// TIA Portal V18 export
VAR_GLOBAL   // PLC tag table "Cabinet_1"
   Sz1_Button_LED_ST25_ST26 AT %Q1100.0 : Bool;
   Sz1_Button_LED_ST26_ST27 AT %Q1100.1 : Bool;
   Sz1_Button_LED_ST24_ST23 AT %Q1100.2 : Bool;
   Sz1_Button_LED_ST23_ST22 AT %Q1100.3 : Bool;
   Sz1_Button_LED_Hyd_Up AT %Q1100.4 : Bool;
   Sz1_Button_LED_Hyd_Down AT %Q1100.5 : Bool;
   Sz1_Button_LED_Air_Up AT %Q1100.6 : Bool;
   Sz1_Button_LED_Air_Down AT %Q1100.7 : Bool;
   Sz1_Button_LED_Wibration AT %Q1101.0 : Bool;
   Sz1_Button_LED_SS_Down AT %Q1101.1 : Bool;
   Sz1_Button_LED_SS_Up AT %Q1101.2 : Bool;
   Sz1_Button_LED_SS_Drive_ST25 AT %Q1101.3 : Bool;
   Sz1_Button_LED_SS_Drive_ST24 AT %Q1101.4 : Bool;
   Sz1_Button_LED_SS_Drive_ST17 AT %Q1101.5 : Bool;
   Sz1_Button_LED_SS_Drive_ST14 AT %Q1101.6 : Bool;
   Reserved AT %Q1101.7 : Bool;
   Sz1_St25_SenA AT %I1100.0 : Bool;
   Sz1_St25_SenB AT %I1100.1 : Bool;
   Sz1_St25_SenC AT %I1100.2 : Bool;
   Sz1_St25_SenD AT %I1100.3 : Bool;
   Sz1_St26_SenA AT %I1100.4 : Bool;
   Sz1_St26_SenB AT %I1100.5 : Bool;
   Sz1_St26_SenC AT %I1100.6 : Bool;
   Sz1_St26_SenD AT %I1100.7 : Bool;
   Sz1_St23_SenA AT %I1101.0 : Bool;
   Sz1_St23_SenB AT %I1101.1 : Bool;
   Sz1_St23_SenC AT %I1101.2 : Bool;
   Sz1_St23_SenD AT %I1101.3 : Bool;
   Sz1_St24_SenA AT %I1101.4 : Bool;
   Sz1_St24_SenB AT %I1101.5 : Bool;
   Sz1_St24_SenC AT %I1101.6 : Bool;
   Sz1_St24_SenD AT %I1101.7 : Bool;
   Sz1_Button_ST25_ST26 AT %I1102.0 : Bool;
   Sz1_Button_ST26_ST27 AT %I1102.1 : Bool;
   Sz1_Button_ST24_ST23 AT %I1102.2 : Bool;
   Sz1_Button_ST23_ST22 AT %I1102.3 : Bool;
   Sz1_Button_Hyd_Up AT %I1102.4 : Bool;
   Sz1_Button_Hyd_Down AT %I1102.5 : Bool;
   Sz1_Button_Air_Up AT %I1102.6 : Bool;
   Sz1_Button_Air_Down AT %I1102.7 : Bool;
   Sz1_Button_Wibration AT %I1103.0 : Bool;
   Sz1_Button_SS_Down AT %I1103.1 : Bool;
   Sz1_Button_SS_Up AT %I1103.2 : Bool;
   Sz1_Button_SS_Drive_ST25 AT %I1103.3 : Bool;
   Sz1_Button_SS_Drive_ST24 AT %I1103.4 : Bool;
   Sz1_Button_SS_Drive_ST17 AT %I1103.5 : Bool;
   Sz1_Button_SS_Drive_ST14 AT %I1103.6 : Bool;
   "Reserved(1)" AT %I1103.7 : Bool;
   Sz1_Button_Wib_ST25 AT %I1104.0 : Bool;
   Sz1_Button_Wib_ST24 AT %I1104.1 : Bool;
   Sz1_Button_Wib_ST23 AT %I1104.2 : Bool;
   Sz1_Button_Centering_ST23 AT %I1104.3 : Bool;
   Sz1_Button_Centering_ST22 AT %I1104.4 : Bool;
   "Reserved(2)" AT %I1104.5 : Bool;
   "Reserved(3)" AT %I1104.6 : Bool;
   "Reserved(4)" AT %I1104.7 : Bool;
   Sz1_Button_LED_Centering_ST23 AT %Q1102.0 : Bool;
   Sz1_Button_LED_Centering_ST22 AT %Q1102.1 : Bool;
   "Reserved(5)" AT %Q1102.2 : Bool;
   "Reserved(6)" AT %Q1102.3 : Bool;
   "Reserved(7)" AT %Q1102.4 : Bool;
   "Reserved(8)" AT %Q1102.5 : Bool;
   "Reserved(9)" AT %Q1102.6 : Bool;
   "Reserved(10)" AT %Q1102.7 : Bool;
   Sz1_Safety1_1 AT %I1150.0 : Bool;
   "Reserved(11)" AT %I1150.1 : Bool;
   "Reserved(12)" AT %I1150.2 : Bool;
   "Reserved(13)" AT %I1150.3 : Bool;
   Sz1_Safety1_2 AT %I1150.4 : Bool;
   "Reserved(14)" AT %I1150.5 : Bool;
   "Reserved(15)" AT %I1150.6 : Bool;
   "Reserved(16)" AT %I1150.7 : Bool;
   "Reserved(17)" AT %I1151.0 : Bool;
   "Reserved(18)" AT %I1151.1 : Bool;
   "Reserved(19)" AT %I1151.2 : Bool;
   "Reserved(20)" AT %I1151.3 : Bool;
   "Reserved(21)" AT %I1151.4 : Bool;
   "Reserved(22)" AT %I1151.5 : Bool;
   "Reserved(23)" AT %I1151.6 : Bool;
   "Reserved(24)" AT %I1151.7 : Bool;
END_VAR
